// TIA Portal project "TIA_Python_TCP_y" (V19)

(* hardware
DEVICE "S7-1500/ET200MP station_1"  S7-1500 station
   slot 0: "Rail_0"  Rack  6ES7 590-1***0-0AA0
   slot 1: "PLC_1"  CPU 1511-1 PN  6ES7 511-1AL03-0AB0  V3.1
      slot 3: "CPU display_1"  6ES7591-1AA00-0AA0
      slot 32768: "PROFINET interface_1"  X1
         slot 32769: "Port_1"  X1 P1
         slot 32770: "Port_2"  X1 P2
      slot 34817: "Virtual CP interface port_1"  Virtual CP interface port  Virtual CP interface port
*)

// ===== PLC "PLC_1"  CPU 1511-1 PN =====

VAR_GLOBAL   // PLC tag table "Default tag table"
   "Tag_1" AT %M0.0 : Bool;
   "Tag_2" AT %M10.0 : Bool;
END_VAR

// folder: 03-Data

DATA_BLOCK "DB_Product"   // DB1
{ S7_Optimized_Access := 'TRUE' }
VERSION : 0.1
   VAR
      Activate : Bool;
      ProductID : String[12] := '000000000001';
      Weight : Int := 125;
      PrinterNo : USInt := 1;
      LabalStatus : USInt;
   END_VAR
BEGIN
END_DATA_BLOCK

DATA_BLOCK "DB_Communication"   // DB2
{ S7_Optimized_Access := 'TRUE' }
VERSION : 0.1
   VAR
      Connected : Bool;
      TxRequest : Bool;
      TxBusy : Bool;
      TxDone : Bool;
      RxNew : Bool;
      CommError : Bool;
      TxCount : DInt;
      RxCount : DInt;
      LastTxID : String[4];
      LastRxID : String[4];
      LastTxTest : String[80];
      LastRxTest : String[80];
      TxBuffer : Array[0..239] of Byte;
      RxBuffer : Array[0..239] of Byte;
      Enable : Bool;
      ConnParam : TCON_IP_v4;
      TconDone : Bool;
      TconBusy : Bool;
      TconError : Bool;
      TconStatus : Word;
      Req_RW01 : Bool;
      Req_RG01 : Bool;
      Req_RE01 : Bool;
      TxError : Bool;
      TxStatus : Word;
      RxBusy : Bool;
      RxError : Bool;
      RxStatus : Word;
      RxLength : UDInt;
      MW01_Received : Bool;
      MG01_Received : Bool;
      ME01_Received : Bool;
      TdisDone : Bool;
      TdisBusy : Bool;
      TdisError : Bool;
      TdisStatus : Word;
      SeqInit : Bool;
      TestErrorLatched : Bool;
      TestStatus : Word;
      TestTconStatus : Word;
      TconErrorLatched : Bool;
      MW01_Received_Latched : Bool;
      MG01_Received_Latched : Bool;
      ME01_Received_Latched : Bool;
      Sequance_Start : Bool;
   END_VAR
BEGIN
   ConnParam.ID := 1;
   ConnParam.ActiveEstablished := 1;
   ConnParam.RemoteAddress.ADDR[1] := 192;
   ConnParam.RemoteAddress.ADDR[2] := 168;
   ConnParam.RemotePort := 2000;
   ConnParam.RemoteAddress.ADDR[3] := 50;
   ConnParam.RemoteAddress.ADDR[4] := 1;
END_DATA_BLOCK

DATA_BLOCK "DB_TCP_Client"   // DB4
{ S7_Optimized_Access := 'TRUE' }
VERSION : 0.1
// stored: InstanceOfName FB_TCP_Client
"FB_TCP_Client"
BEGIN
END_DATA_BLOCK

DATA_BLOCK "DB_FB_Sequance"   // DB7
{ S7_Optimized_Access := 'TRUE' }
VERSION : 0.1
// stored: InstanceOfName FB_Sequance
"FB_Sequance"
BEGIN
END_DATA_BLOCK

// folder: (top level)

ORGANIZATION_BLOCK "Main"   // OB1, LAD, ProgramCycle
TITLE = "Main Program Sweep (Cycle)"
{ S7_Optimized_Access := 'TRUE' }
VERSION : 0.1
   VAR_INPUT
      Initial_Call : Bool;   // Initial call of this OB
      Remanence : Bool;   // =True, if remanent data are available
   END_VAR
BEGIN

REGION Network 1
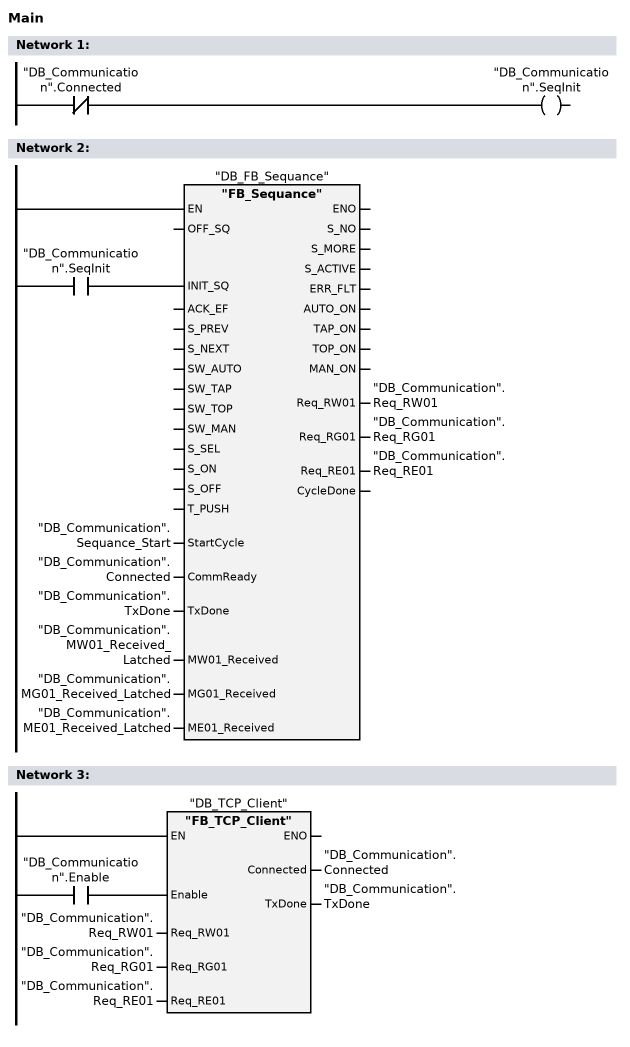
   RUNG wire#powerrail
      I_Contact( "DB_Communication".Connected )
      Coil( "DB_Communication".SeqInit )
   END_RUNG
   // the same network as SCL:
   "DB_Communication".SeqInit := NOT "DB_Communication".Connected;
END_REGION

REGION Network 2
   RUNG wire#powerrail
      "DB_FB_Sequance"(INIT_SQ := wire#w1, OFF_SQ :=, ACK_EF :=, S_PREV :=, S_NEXT :=, SW_AUTO :=, SW_TAP :=, SW_TOP :=, SW_MAN :=, S_SEL :=, S_ON :=, S_OFF :=, T_PUSH :=, StartCycle := "DB_Communication".Sequance_Start, CommReady := "DB_Communication".Connected, TxDone := "DB_Communication".TxDone, MW01_Received := "DB_Communication".MW01_Received_Latched, MG01_Received := "DB_Communication".MG01_Received_Latched, ME01_Received := "DB_Communication".ME01_Received_Latched, S_NO =>, S_MORE =>, S_ACTIVE =>, ERR_FLT =>, AUTO_ON =>, TAP_ON =>, TOP_ON =>, MAN_ON =>, Req_RW01 => "DB_Communication".Req_RW01, Req_RG01 => "DB_Communication".Req_RG01, Req_RE01 => "DB_Communication".Req_RE01, CycleDone =>)
   END_RUNG
   RUNG wire#powerrail
      Contact( "DB_Communication".SeqInit )
   END_RUNG wire#w1
   // the same network as SCL:
   "DB_FB_Sequance"(INIT_SQ := "DB_Communication".SeqInit,   // "FB_Sequance"
                    StartCycle := "DB_Communication".Sequance_Start,
                    CommReady := "DB_Communication".Connected,
                    TxDone := "DB_Communication".TxDone,
                    MW01_Received := "DB_Communication".MW01_Received_Latched,
                    MG01_Received := "DB_Communication".MG01_Received_Latched,
                    ME01_Received := "DB_Communication".ME01_Received_Latched,
                    Req_RW01 => "DB_Communication".Req_RW01,
                    Req_RG01 => "DB_Communication".Req_RG01,
                    Req_RE01 => "DB_Communication".Req_RE01);
END_REGION

REGION Network 3
   RUNG wire#powerrail
      "DB_TCP_Client"(Enable := wire#w1, Req_RW01 := "DB_Communication".Req_RW01, Req_RG01 := "DB_Communication".Req_RG01, Req_RE01 := "DB_Communication".Req_RE01, Connected => "DB_Communication".Connected, TxDone => "DB_Communication".TxDone)
   END_RUNG
   RUNG wire#powerrail
      Contact( "DB_Communication".Enable )
   END_RUNG wire#w1
   // the same network as SCL:
   "DB_TCP_Client"(Enable := "DB_Communication".Enable,   // "FB_TCP_Client"
                   Req_RW01 := "DB_Communication".Req_RW01,
                   Req_RG01 := "DB_Communication".Req_RG01,
                   Req_RE01 := "DB_Communication".Req_RE01,
                   Connected => "DB_Communication".Connected,
                   TxDone => "DB_Communication".TxDone);
END_REGION

REGION Network 4: Set sequence to initial state
END_REGION
END_ORGANIZATION_BLOCK

// folder: 01-Sequance

FUNCTION_BLOCK "FB_Sequance"   // FB1, GRAPH_PLUS
{ S7_Optimized_Access := 'TRUE' }
VERSION : 0.1
   VAR_INPUT
      OFF_SQ : Bool := false;   // Turn sequence off
      INIT_SQ : Bool := false;   // Set sequence to initial state
      ACK_EF : Bool := false;   // Acknowledge all errors and faults
      S_PREV : Bool := false;   // Output previous step in parameter S_NO
      S_NEXT : Bool := false;   // Indicate next step in parameter S_NO
      SW_AUTO : Bool := false;   // Automatic mode
      SW_TAP : Bool := false;   // Semiautomatic/switch with transition
      SW_TOP : Bool := false;   // Semiautomatic/ignore transition
      SW_MAN : Bool := false;   // Manual mode
      S_SEL : Int := 0;   // Select step to be output to S_NO
      S_ON : Bool := false;   // Activate step indicated in S_NO
      S_OFF : Bool := false;   // Disable step indicated in S_NO
      T_PUSH : Bool := false;   // Enable transition to switch in semi automatic mode
      StartCycle : Bool;
      CommReady : Bool;
      TxDone : Bool;
      MW01_Received : Bool;
      MG01_Received : Bool;
      ME01_Received : Bool;
   END_VAR
   VAR_OUTPUT
      S_NO : Int := 0;   // Step number
      S_MORE : Bool := false;   // More steps are available and can be shown in S_NO
      S_ACTIVE : Bool := false;   // Step indicated in S_NO is active
      ERR_FLT : Bool := false;   // Interlock or supervision group error
      AUTO_ON : Bool := false;   // Automatic mode is active
      TAP_ON : Bool := false;   // Semiautomatic mode/step with transition enabled
      TOP_ON : Bool := false;   // Semiautomatic mode/ignore transition enabled
      MAN_ON : Bool := false;   // Manual mode is active
      Req_RW01 : Bool;
      Req_RG01 : Bool;
      Req_RE01 : Bool;
      CycleDone : Bool;
   END_VAR
   VAR
      HMI_INFO : Array[0..8] of UInt;
      IF_PAR : G7_IfParPlus_V6;
      RT_DATA : G7_RTDataPlus_V6;   // Internal data area
      Trans1 : G7_TransitionPlus_V6;   // Transition structure
      Trans2 : G7_TransitionPlus_V6;   // Transition structure
      Trans3 : G7_TransitionPlus_V6;   // Transition structure
      Trans4 : G7_TransitionPlus_V6;   // Transition structure
      Trans5 : G7_TransitionPlus_V6;   // Transition structure
      Trans6 : G7_TransitionPlus_V6;   // Transition structure
      Trans7 : G7_TransitionPlus_V6;   // Transition structure
      Trans8 : G7_TransitionPlus_V6;   // Transition structure
      Trans9 : G7_TransitionPlus_V6;   // Transition structure
      Trans10 : G7_TransitionPlus_V6;   // Transition structure
      IDLE : G7_StepPlus_V6;   // Step structure
      SEND_RW01 : G7_StepPlus_V6;   // Step structure
      WAIT_MW01 : G7_StepPlus_V6;   // Step structure
      MOVE_TO_SCALE : G7_StepPlus_V6;   // Step structure
      SEND_RG01 : G7_StepPlus_V6;   // Step structure
      WAIT_MG01 : G7_StepPlus_V6;   // Step structure
      MOVE_TO_LABEL : G7_StepPlus_V6;   // Step structure
      SEND_RE01 : G7_StepPlus_V6;   // Step structure
      WAIT_ME01 : G7_StepPlus_V6;   // Step structure
      COMPLETE : G7_StepPlus_V6;   // Step structure
      SINI : Array[0..1] of USInt;
      LSTT : Array[0..9] of USInt;
      ATAJ : Array[0..9] of USInt;
      ATAB : Array[0..9] of USInt;
      PSTT : Array[0..9] of USInt;
      NSTT : Array[0..9] of USInt;
      ASSJ : Array[0..9] of USInt;
      ASSB : Array[0..9] of USInt;
      PTTS : Array[0..9] of USInt;
      NTTS : Array[0..9] of USInt;
      SW_SQTS : Array[0..9] of USInt;
      SWITCH : Array[0..0] of USInt;
      TVX : Array[0..1] of USInt;
      TTX : Array[0..1] of USInt;
      TSX : Array[0..1] of USInt;
      S00X : Array[0..1] of USInt;
      SOFFX : Array[0..1] of USInt;
      SONX : Array[0..1] of USInt;
      SAX : Array[0..1] of USInt;
      SERRX : Array[0..10] of USInt;
      SMX : Array[0..10] of USInt;
      S0X : Array[0..10] of USInt;
      S1X : Array[0..10] of USInt;
      IL_ALARM_INST : Diag_Alarm;
      SUP_ALARM_INST : Diag_Alarm;
      STEP_TIME_ALARM_INST : Diag_Alarm;
      IEC_TIMER_INST : IEC_TIMER;
      TRANSACTION_FLAG : Bool := false;
   END_VAR
   // SINI[0] := 2;
   // LSTT[0] := 255;
   // LSTT[1] := 255;
   // LSTT[2] := 255;
   // LSTT[3] := 255;
   // LSTT[4] := 255;
   // LSTT[5] := 255;
   // LSTT[6] := 255;
   // LSTT[7] := 255;
   // LSTT[8] := 255;
   // ATAJ[1] := 1;
   // ATAJ[2] := 2;
   // ATAJ[3] := 3;
   // ATAJ[4] := 4;
   // ATAJ[5] := 5;
   // ATAJ[6] := 6;
   // ATAJ[7] := 7;
   // ATAJ[8] := 8;
   // ATAJ[9] := 9;
   // ATAB[1] := 1;
   // ATAB[2] := 2;
   // ATAB[3] := 3;
   // ATAB[4] := 4;
   // ATAB[5] := 5;
   // ATAB[6] := 6;
   // ATAB[7] := 7;
   // ATAB[8] := 8;
   // ATAB[9] := 9;
   // PSTT[1] := 1;
   // PSTT[2] := 2;
   // PSTT[3] := 3;
   // PSTT[4] := 4;
   // PSTT[5] := 5;
   // PSTT[6] := 6;
   // PSTT[7] := 7;
   // PSTT[8] := 8;
   // PSTT[9] := 9;
   // NSTT[0] := 1;
   // NSTT[1] := 2;
   // NSTT[2] := 3;
   // NSTT[3] := 4;
   // NSTT[4] := 5;
   // NSTT[5] := 6;
   // NSTT[6] := 7;
   // NSTT[7] := 8;
   // NSTT[8] := 9;
   // ASSJ[1] := 1;
   // ASSJ[2] := 2;
   // ASSJ[3] := 3;
   // ASSJ[4] := 4;
   // ASSJ[5] := 5;
   // ASSJ[6] := 6;
   // ASSJ[7] := 7;
   // ASSJ[8] := 8;
   // ASSJ[9] := 9;
   // ASSB[1] := 1;
   // ASSB[2] := 2;
   // ASSB[3] := 3;
   // ASSB[4] := 4;
   // ASSB[5] := 5;
   // ASSB[6] := 6;
   // ASSB[7] := 7;
   // ASSB[8] := 8;
   // ASSB[9] := 9;
   // PTTS[0] := 255;
   // PTTS[2] := 1;
   // PTTS[3] := 2;
   // PTTS[4] := 3;
   // PTTS[5] := 4;
   // PTTS[6] := 5;
   // PTTS[7] := 6;
   // PTTS[8] := 7;
   // PTTS[9] := 8;
   // NTTS[1] := 1;
   // NTTS[2] := 2;
   // NTTS[3] := 3;
   // NTTS[4] := 4;
   // NTTS[5] := 5;
   // NTTS[6] := 6;
   // NTTS[7] := 7;
   // NTTS[8] := 8;
   // NTTS[9] := 9;
   // TVX[0] := 16#1;
   // TTX[0] := 16#1;
   // TSX[0] := 16#1;
   // S00X[0] := 16#1;
   // SOFFX[0] := 16#1;
   // SONX[0] := 16#1;
   // SAX[0] := 16#1;
   // SERRX[0] := 16#1;
   // SMX[0] := 16#1;
   // S0X[0] := 16#1;
   // S1X[0] := 16#1;
BEGIN
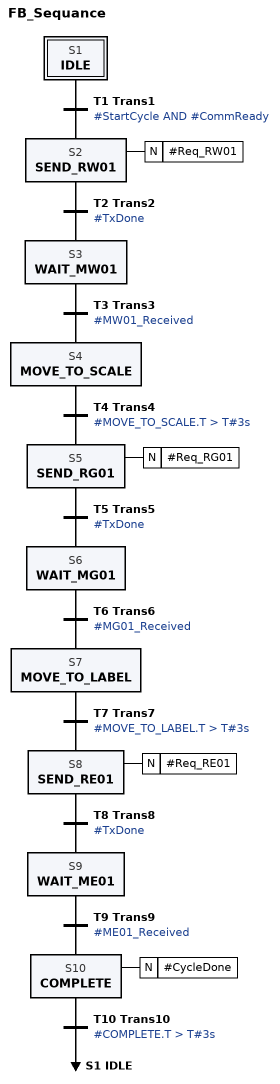
   // sequencer 1
   INITIAL_STEP IDLE:   // S1, max time T#10S, warning time T#7S
   END_STEP
   TRANSITION Trans1 FROM IDLE TO SEND_RW01   // T1
      := #StartCycle AND #CommReady;
   END_TRANSITION
   STEP SEND_RW01:   // S2, max time T#10S, warning time T#7S
              N    #Req_RW01
   END_STEP
   TRANSITION Trans2 FROM SEND_RW01 TO WAIT_MW01   // T2
      := #TxDone;
   END_TRANSITION
   STEP WAIT_MW01:   // S3, max time T#10S, warning time T#7S
   END_STEP
   TRANSITION Trans3 FROM WAIT_MW01 TO MOVE_TO_SCALE   // T3
      := #MW01_Received;
   END_TRANSITION
   STEP MOVE_TO_SCALE:   // S4, max time T#10S, warning time T#7S
   END_STEP
   TRANSITION Trans4 FROM MOVE_TO_SCALE TO SEND_RG01   // T4
      := #MOVE_TO_SCALE.T > T#3s;
   END_TRANSITION
   STEP SEND_RG01:   // S5, max time T#10S, warning time T#7S
              N    #Req_RG01
   END_STEP
   TRANSITION Trans5 FROM SEND_RG01 TO WAIT_MG01   // T5
      := #TxDone;
   END_TRANSITION
   STEP WAIT_MG01:   // S6, max time T#10S, warning time T#7S
   END_STEP
   TRANSITION Trans6 FROM WAIT_MG01 TO MOVE_TO_LABEL   // T6
      := #MG01_Received;
   END_TRANSITION
   STEP MOVE_TO_LABEL:   // S7, max time T#10S, warning time T#7S
   END_STEP
   TRANSITION Trans7 FROM MOVE_TO_LABEL TO SEND_RE01   // T7
      := #MOVE_TO_LABEL.T > T#3s;
   END_TRANSITION
   STEP SEND_RE01:   // S8, max time T#10S, warning time T#7S
              N    #Req_RE01
   END_STEP
   TRANSITION Trans8 FROM SEND_RE01 TO WAIT_ME01   // T8
      := #TxDone;
   END_TRANSITION
   STEP WAIT_ME01:   // S9, max time T#10S, warning time T#7S
   END_STEP
   TRANSITION Trans9 FROM WAIT_ME01 TO COMPLETE   // T9
      := #ME01_Received;
   END_TRANSITION
   STEP COMPLETE:   // S10, max time T#10S, warning time T#7S
              N    #CycleDone
   END_STEP
   TRANSITION Trans10 FROM COMPLETE TO IDLE   // T10, jump
      := #COMPLETE.T > T#3s;
   END_TRANSITION
END_FUNCTION_BLOCK

// folder: 02-Communication

FUNCTION_BLOCK "FB_TCP_Client"   // FB2, LAD
{ S7_Optimized_Access := 'TRUE' }
VERSION : 0.1
   VAR_INPUT
      Enable : Bool;
      Req_RW01 : Bool;
      Req_RG01 : Bool;
      Req_RE01 : Bool;
   END_VAR
   VAR_OUTPUT
      Connected : Bool;
      TxDone : Bool;
   END_VAR
   VAR
      ConnectTrig : R_TRIG;
      DisconnectTrig : F_TRIG;
      TconErrorLatched : Bool;
      LastTconErrorStatus : Word;
      CommArmed : Bool;
      SendTrig : R_TRIG;
   END_VAR
   VAR_TEMP
      Edge_Memory : Bool;
   END_VAR
BEGIN

REGION Network 1
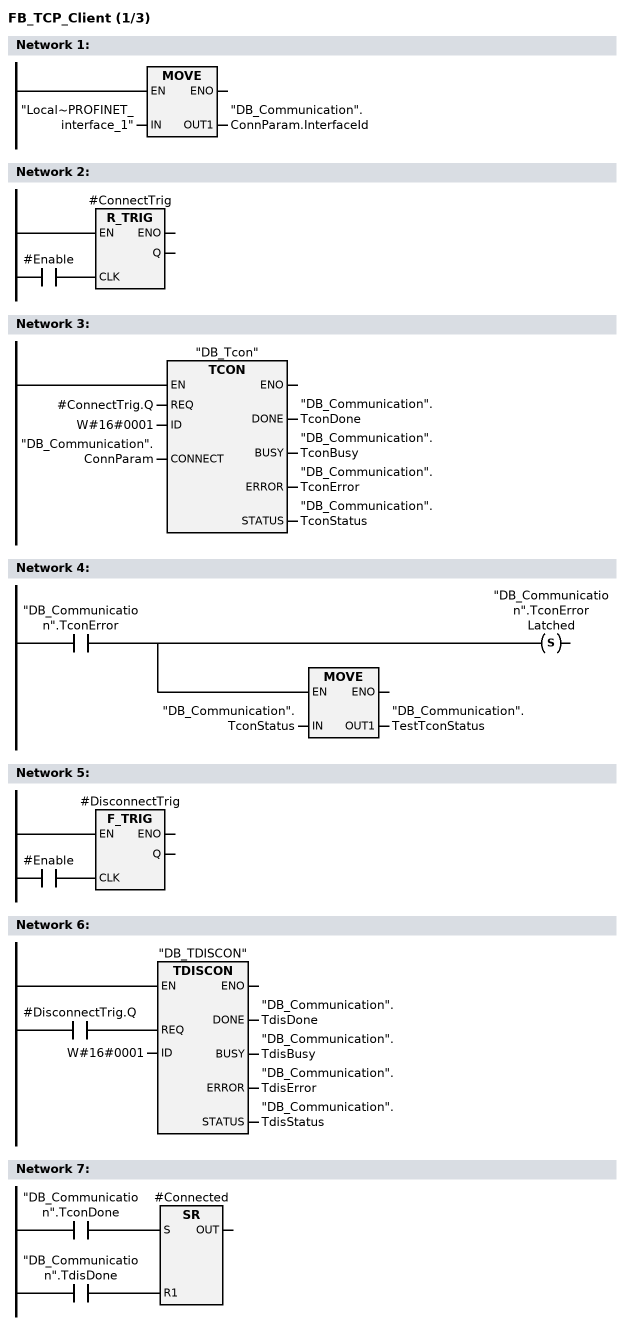
   RUNG wire#powerrail
      Move(in := "Local~PROFINET_interface_1", out1 => "DB_Communication".ConnParam.InterfaceId)
   END_RUNG
   // the same network as SCL:
   "DB_Communication".ConnParam.InterfaceId := "Local~PROFINET_interface_1";
END_REGION

REGION Network 2
   #ConnectTrig(CLK := #Enable);   // R_TRIG
END_REGION

REGION Network 3
   "DB_Tcon"(REQ := #ConnectTrig.Q,   // TCON
             ID := W#16#0001,
             CONNECT := "DB_Communication".ConnParam,
             DONE => "DB_Communication".TconDone,
             BUSY => "DB_Communication".TconBusy,
             ERROR => "DB_Communication".TconError,
             STATUS => "DB_Communication".TconStatus);
END_REGION

REGION Network 4
   RUNG wire#powerrail
      Contact( "DB_Communication".TconError )
      wire#w1
      S_Coil( "DB_Communication".TconErrorLatched )
   END_RUNG
   RUNG wire#w1
      Move(in := "DB_Communication".TconStatus, out1 => "DB_Communication".TestTconStatus)
   END_RUNG
   // the same network as SCL:
   IF "DB_Communication".TconError THEN
       "DB_Communication".TconErrorLatched := TRUE;
       "DB_Communication".TestTconStatus := "DB_Communication".TconStatus;
   END_IF;
END_REGION

REGION Network 5
   #DisconnectTrig(CLK := #Enable);   // F_TRIG
END_REGION

REGION Network 6
   "DB_TDISCON"(REQ := #DisconnectTrig.Q,   // TDISCON
                ID := W#16#0001,
                DONE => "DB_Communication".TdisDone,
                BUSY => "DB_Communication".TdisBusy,
                ERROR => "DB_Communication".TdisError,
                STATUS => "DB_Communication".TdisStatus);
END_REGION

REGION Network 7
   RUNG wire#powerrail
      Contact( "DB_Communication".TconDone )
      S_SR(operand := #Connected, r1 := wire#w1)
   END_RUNG
   RUNG wire#powerrail
      Contact( "DB_Communication".TdisDone )
   END_RUNG wire#w1
   // the same network as SCL:
   IF "DB_Communication".TconDone THEN
       #Connected := TRUE;   // SR flip-flop
   END_IF;
   IF "DB_Communication".TdisDone THEN #Connected := FALSE; END_IF;
END_REGION

REGION Network 8
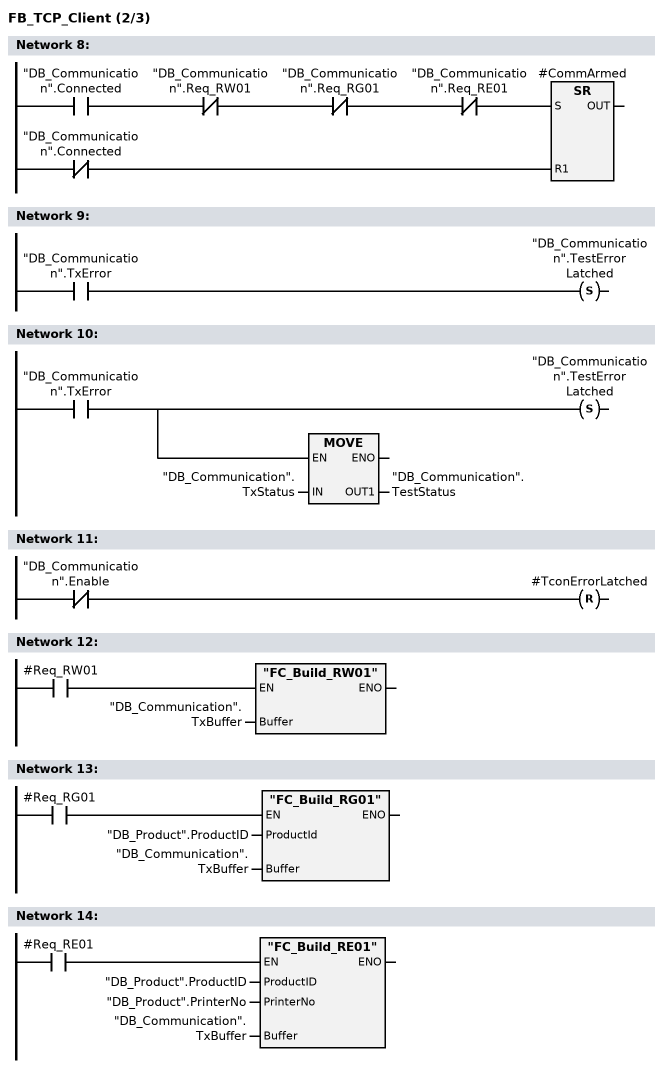
   RUNG wire#powerrail
      Contact( "DB_Communication".Connected )
      I_Contact( "DB_Communication".Req_RW01 )
      I_Contact( "DB_Communication".Req_RG01 )
      I_Contact( "DB_Communication".Req_RE01 )
      S_SR(operand := #CommArmed, r1 := wire#w1)
   END_RUNG
   RUNG wire#powerrail
      I_Contact( "DB_Communication".Connected )
   END_RUNG wire#w1
   // the same network as SCL:
   IF "DB_Communication".Connected AND NOT "DB_Communication".Req_RW01 AND NOT "DB_Communication".Req_RG01 AND NOT "DB_Communication".Req_RE01 THEN
       #CommArmed := TRUE;   // SR flip-flop
   END_IF;
   IF NOT "DB_Communication".Connected THEN #CommArmed := FALSE; END_IF;
END_REGION

REGION Network 9
   RUNG wire#powerrail
      Contact( "DB_Communication".TxError )
      S_Coil( "DB_Communication".TestErrorLatched )
   END_RUNG
   // the same network as SCL:
   IF "DB_Communication".TxError THEN "DB_Communication".TestErrorLatched := TRUE; END_IF;
END_REGION

REGION Network 10
   RUNG wire#powerrail
      Contact( "DB_Communication".TxError )
      wire#w1
      S_Coil( "DB_Communication".TestErrorLatched )
   END_RUNG
   RUNG wire#w1
      Move(in := "DB_Communication".TxStatus, out1 => "DB_Communication".TestStatus)
   END_RUNG
   // the same network as SCL:
   IF "DB_Communication".TxError THEN
       "DB_Communication".TestErrorLatched := TRUE;
       "DB_Communication".TestStatus := "DB_Communication".TxStatus;
   END_IF;
END_REGION

REGION Network 11
   RUNG wire#powerrail
      I_Contact( "DB_Communication".Enable )
      R_Coil( #TconErrorLatched )
   END_RUNG
   // the same network as SCL:
   IF NOT "DB_Communication".Enable THEN #TconErrorLatched := FALSE; END_IF;
END_REGION

REGION Network 12
   RUNG wire#powerrail
      Contact( #Req_RW01 )
      "FC_Build_RW01"(Buffer := "DB_Communication".TxBuffer)
   END_RUNG
   // the same network as SCL:
   IF #Req_RW01 THEN "FC_Build_RW01"(Buffer := "DB_Communication".TxBuffer); END_IF;
END_REGION

REGION Network 13
   RUNG wire#powerrail
      Contact( #Req_RG01 )
      "FC_Build_RG01"(ProductId := "DB_Product".ProductID, Buffer := "DB_Communication".TxBuffer)
   END_RUNG
   // the same network as SCL:
   IF #Req_RG01 THEN
       "FC_Build_RG01"(ProductId := "DB_Product".ProductID, Buffer := "DB_Communication".TxBuffer);
   END_IF;
END_REGION

REGION Network 14
   RUNG wire#powerrail
      Contact( #Req_RE01 )
      "FC_Build_RE01"(ProductID := "DB_Product".ProductID, PrinterNo := "DB_Product".PrinterNo, Buffer := "DB_Communication".TxBuffer)
   END_RUNG
   // the same network as SCL:
   IF #Req_RE01 THEN
       "FC_Build_RE01"(ProductID := "DB_Product".ProductID,
                       PrinterNo := "DB_Product".PrinterNo,
                       Buffer := "DB_Communication".TxBuffer);
   END_IF;
END_REGION

REGION Network 15
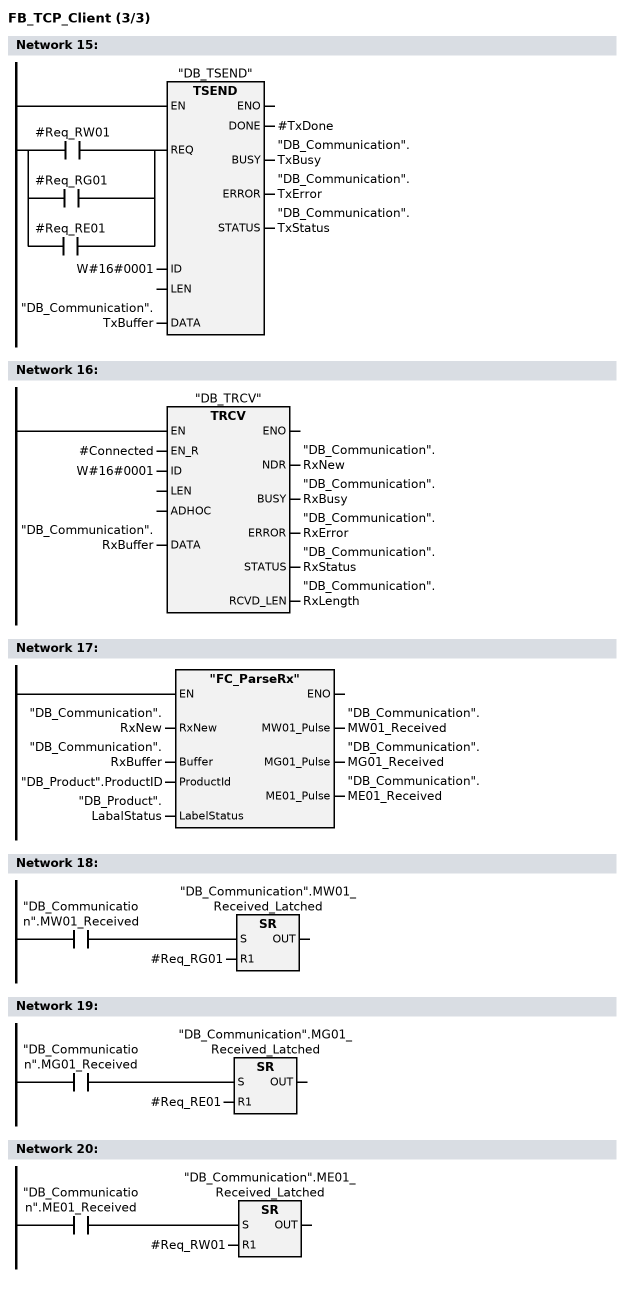
   "DB_TSEND"(REQ := #Req_RW01 OR #Req_RG01 OR #Req_RE01,   // TSEND
              ID := W#16#0001,
              DATA := "DB_Communication".TxBuffer,
              DONE => #TxDone,
              BUSY => "DB_Communication".TxBusy,
              ERROR => "DB_Communication".TxError,
              STATUS => "DB_Communication".TxStatus);
END_REGION

REGION Network 16
   "DB_TRCV"(EN_R := #Connected,   // TRCV
             ID := W#16#0001,
             DATA := "DB_Communication".RxBuffer,
             NDR => "DB_Communication".RxNew,
             BUSY => "DB_Communication".RxBusy,
             ERROR => "DB_Communication".RxError,
             STATUS => "DB_Communication".RxStatus,
             RCVD_LEN => "DB_Communication".RxLength);
END_REGION

REGION Network 17
   RUNG wire#powerrail
      "FC_ParseRx"(RxNew := "DB_Communication".RxNew, Buffer := "DB_Communication".RxBuffer, ProductId := "DB_Product".ProductID, LabelStatus := "DB_Product".LabalStatus, MW01_Pulse => "DB_Communication".MW01_Received, MG01_Pulse => "DB_Communication".MG01_Received, ME01_Pulse => "DB_Communication".ME01_Received)
   END_RUNG
   // the same network as SCL:
   "FC_ParseRx"(RxNew := "DB_Communication".RxNew,
                Buffer := "DB_Communication".RxBuffer,
                ProductId := "DB_Product".ProductID,
                LabelStatus := "DB_Product".LabalStatus,
                MW01_Pulse => "DB_Communication".MW01_Received,
                MG01_Pulse => "DB_Communication".MG01_Received,
                ME01_Pulse => "DB_Communication".ME01_Received);
END_REGION

REGION Network 18
   RUNG wire#powerrail
      Contact( "DB_Communication".MW01_Received )
      S_SR(operand := "DB_Communication".MW01_Received_Latched, r1 := #Req_RG01)
   END_RUNG
   // the same network as SCL:
   IF "DB_Communication".MW01_Received THEN
       "DB_Communication".MW01_Received_Latched := TRUE;   // SR flip-flop
   END_IF;
   IF #Req_RG01 THEN "DB_Communication".MW01_Received_Latched := FALSE; END_IF;
END_REGION

REGION Network 19
   RUNG wire#powerrail
      Contact( "DB_Communication".MG01_Received )
      S_SR(operand := "DB_Communication".MG01_Received_Latched, r1 := #Req_RE01)
   END_RUNG
   // the same network as SCL:
   IF "DB_Communication".MG01_Received THEN
       "DB_Communication".MG01_Received_Latched := TRUE;   // SR flip-flop
   END_IF;
   IF #Req_RE01 THEN "DB_Communication".MG01_Received_Latched := FALSE; END_IF;
END_REGION

REGION Network 20
   RUNG wire#powerrail
      Contact( "DB_Communication".ME01_Received )
      S_SR(operand := "DB_Communication".ME01_Received_Latched, r1 := #Req_RW01)
   END_RUNG
   // the same network as SCL:
   IF "DB_Communication".ME01_Received THEN
       "DB_Communication".ME01_Received_Latched := TRUE;   // SR flip-flop
   END_IF;
   IF #Req_RW01 THEN "DB_Communication".ME01_Received_Latched := FALSE; END_IF;
END_REGION
END_FUNCTION_BLOCK

FUNCTION "FC_Build_RW01" : Void   // FC1, SCL
{ S7_Optimized_Access := 'TRUE' }
VERSION : 0.1
   VAR_IN_OUT
      Buffer : Array[0..239] of Byte;
   END_VAR
   VAR_TEMP
      i : Int;
   END_VAR
BEGIN
   // Fill complete telegram with ASCII spaces
   FOR #i := 0 TO 239 DO
       #Buffer[#i] := 16#20;
   END_FOR;

   // STX
   #Buffer[0] := 16#02;

   // "RW01"
   #Buffer[1] := 16#52;    // R
   #Buffer[2] := 16#57;    // W
   #Buffer[3] := 16#30;    // 0
   #Buffer[4] := 16#31;    // 1

   // |
   #Buffer[5] := 16#7C;

   // ETX
   #Buffer[239] := 16#03;
END_FUNCTION

FUNCTION "FC_ParseRx" : Void   // FC2, SCL
{ S7_Optimized_Access := 'TRUE' }
VERSION : 0.1
   VAR_INPUT
      RxNew : Bool;
   END_VAR
   VAR_OUTPUT
      MW01_Pulse : Bool;
      MG01_Pulse : Bool;
      ME01_Pulse : Bool;
   END_VAR
   VAR_IN_OUT
      Buffer : Array[0..239] of Byte;
      ProductId : String;
      LabelStatus : USInt;
   END_VAR
   VAR_TEMP
      i : Int;
   END_VAR
BEGIN
   #MW01_Pulse := FALSE;
   #MG01_Pulse := FALSE;
   #ME01_Pulse := FALSE;

   IF #RxNew THEN

       IF (#Buffer[0] = 16#02) AND
           (#Buffer[239] = 16#03) THEN

           // MW01
           IF (#Buffer[1] = 16#4D) AND
               (#Buffer[2] = 16#57) AND
               (#Buffer[3] = 16#30) AND
               (#Buffer[4] = 16#31) THEN

               // 12-character Product ID
               #ProductId := '            ';

               FOR #i := 0 TO 11 DO
                   #ProductId[#i + 1] :=
                   BYTE_TO_CHAR(#Buffer[#i + 6]);
               END_FOR;

               #MW01_Pulse := TRUE;


               // MG01
           ELSIF (#Buffer[1] = 16#4D) AND
               (#Buffer[2] = 16#47) AND
               (#Buffer[3] = 16#30) AND
               (#Buffer[4] = 16#31) THEN

               #MG01_Pulse := TRUE;


               // ME01
           ELSIF (#Buffer[1] = 16#4D) AND
               (#Buffer[2] = 16#45) AND
               (#Buffer[3] = 16#30) AND
               (#Buffer[4] = 16#31) THEN

               IF #Buffer[19] = 16#30 THEN
                   #LabelStatus := 0;

               ELSIF #Buffer[19] = 16#31 THEN
                   #LabelStatus := 1;
               END_IF;

               #ME01_Pulse := TRUE;

           END_IF;

       END_IF;

   END_IF;
END_FUNCTION

FUNCTION "FC_Build_RG01" : Void   // FC3, SCL
{ S7_Optimized_Access := 'TRUE' }
VERSION : 0.1
   VAR_INPUT
      ProductId : String;
   END_VAR
   VAR_IN_OUT
      Buffer : Array[0..239] of Byte;
   END_VAR
   VAR_TEMP
      i : Int;
   END_VAR
BEGIN
   // --------------------------------------------------
   // Clear complete 240 byte telegram with ASCII SPACE
   // --------------------------------------------------

   FOR #i := 0 TO 239 DO
       #Buffer[#i] := 16#20;
   END_FOR;


   // --------------------------------------------------
   // STX
   // --------------------------------------------------

   #Buffer[0] := 16#02;


   // --------------------------------------------------
   // Message ID = RG01
   // --------------------------------------------------

   #Buffer[1] := 16#52;     // R
   #Buffer[2] := 16#47;     // G
   #Buffer[3] := 16#30;     // 0
   #Buffer[4] := 16#31;     // 1


   // --------------------------------------------------
   // Separator |
   // --------------------------------------------------

   #Buffer[5] := 16#7C;


   // --------------------------------------------------
   // Product ID - 12 characters
   // Buffer[6..17]
   // --------------------------------------------------

   FOR #i := 0 TO 11 DO
       #Buffer[#i + 6] := CHAR_TO_BYTE(#ProductId[#i + 1]);
   END_FOR;


   // --------------------------------------------------
   // Separator |
   // --------------------------------------------------

   #Buffer[18] := 16#7C;


   // --------------------------------------------------
   // Fixed weight = 0125 kg
   // --------------------------------------------------

   #Buffer[19] := 16#30;    // 0
   #Buffer[20] := 16#31;    // 1
   #Buffer[21] := 16#32;    // 2
   #Buffer[22] := 16#35;    // 5


   // --------------------------------------------------
   // Separator |
   // --------------------------------------------------

   #Buffer[23] := 16#7C;


   // --------------------------------------------------
   // ETX
   // --------------------------------------------------

   #Buffer[239] := 16#03;
END_FUNCTION

FUNCTION "FC_Build_RE01" : Void   // FC4, SCL
{ S7_Optimized_Access := 'TRUE' }
VERSION : 0.1
   VAR_INPUT
      ProductID : String;
      PrinterNo : USInt;
   END_VAR
   VAR_IN_OUT
      Buffer : Array[0..239] of Byte;
   END_VAR
   VAR_TEMP
      i : Int;
   END_VAR
BEGIN
   // Fill complete telegram with ASCII SPACE
   FOR #i := 0 TO 239 DO
       #Buffer[#i] := 16#20;
   END_FOR;


   // STX
   #Buffer[0] := 16#02;


   // Message ID = RE01
   #Buffer[1] := 16#52;    // R
   #Buffer[2] := 16#45;    // E
   #Buffer[3] := 16#30;    // 0
   #Buffer[4] := 16#31;    // 1


   // |
   #Buffer[5] := 16#7C;


   // Product ID = 12 characters
   FOR #i := 0 TO 11 DO
       #Buffer[#i + 6] := CHAR_TO_BYTE(#ProductID[#i + 1]);
   END_FOR;


   // |
   #Buffer[18] := 16#7C;


   // Printer number
   IF #PrinterNo = 0 THEN
       #Buffer[19] := 16#30;    // "0"
   ELSE
       #Buffer[19] := 16#31;    // "1"
   END_IF;


   // |
   #Buffer[20] := 16#7C;


   // ETX
   #Buffer[239] := 16#03;
END_FUNCTION